PROGRAM MAIN
VAR

END_VAR

// System Control
gvlSystem.iTaskIdx  := GETCURTASKINDEXEX();
prgSystem(iTaskIdx 	:= gvlSystem.iTaskIdx,
	   bFirstCycle  := gvlSystem.bFirstCycle);

// IO (comment for simulation)
//prgIO();
	   
// TCP Connection
prgTCPComm(cmdData => gvlMotion.cmdData);

// Motion Control
prgMotion(
	cmdData:= gvlMotion.cmdData, 
	bAutoEnableDrive:= gvlMotion.bEnableDrive, 
	bAutoStartDrive:= gvlMotion.bStartDrive, 
	bAutoInterlockOK:= gvlMotion.bInterlockOK, 
	bAutoTriggerDefault:= gvlMotion.bTriggerDefault, 
	autoDriveStatus=> gvlMotion.driveStatus, 
	cmdResponse=>, 
	arrServoInterface:= gvlServo.arrServoInterface);

END_PROGRAM

(* stored: Version 1.1.0.1, ProductVersion 3.1.4024.12
   POU MAIN: Id {9767283b-cca1-4624-be02-ae2381d3ffbe}, SpecialFunc None *)
